// TwinCAT 3 PLC project Main
// ProgramVersion: 3.1.4023.0
// libraries:
//   MotorPositionController, * (Randolf)
//   Tc2_MC2, * (Beckhoff Automation GmbH)
//   Tc2_Standard, * (Beckhoff Automation GmbH)
//   Tc2_System, * (Beckhoff Automation GmbH)
//   Tc3_Module, * (Beckhoff Automation GmbH)
//   VisuDialogs, * (System)
//   VisuSymbols,3.5.10.0,System
// project tree:
//   DUTs/ SensorData.TcDUT
//   / GlobalTextList.TcGTLO, PlcTask.TcTTO (not stored), 视图管理器.TcVMO (not stored)
//   GVLs/ GVL.TcGVL
//   POUs/ MAIN.TcPOU
//   VISUs/ Visualization.TcVIS
// real-time tasks:
//   TASK PlcTask: cycle T#1ms, priority 20, ADS port 350
// motion (NC):
//   TASK NC-Task 1 SAF: cycle T#1ms, priority 4, ADS port 501
//   TASK NC-Task 1 SVB: cycle T#1ms, priority 8, ADS port 511
//   AXIS Axis 1 (id 1)
//     General: UnitName=Degree
//     Dynamic: Acceleration=270, Deceleration=270, Jerk=405
//     Velo: RefSearch=180.759448242188, RefSync=180.759448242188, SlowManual=60, FastManual=120, Fast=18075.9448242188, Maximum=360
//     PositionAreaControl: Enable=false
//     TargetPosControl: Enable=false
//     OtherSettings: AllowMotionCmdToSlave=true
//     encoder EncType=8
//       EncPara: ScaleFactorNumerator=360, ScaleFactorDenominator=1048576, MaxCount=#xffffffff
//     drive DrvType=9
//       DrvPara: MaxCount=#xffffffff, DriveControlDWord=#x00030100
//         Analog: VeloReferenz=360, VeloScale=1.02400649589962, TorqueSetpointScale=10, ScaleFactorActTorque=0.1
//         TimeComp: TaskDelayCycles=1
//     controller CtrType=1
//       CtrPara: PriorControlFactor=1
//         PosDiffControl: Enable=false
//         Observer: BandWidth=20
// I/O:
//   DEVICE Device 3 (EtherCAT), AmsNetId 192.168.137.1.4.1
//     Term 1 (EK1100) [EK1100 EtherCAT Coupler (2A E-Bus)]
//       Term 2 (EL9505) [EL9505 Power supply terminal 5V]
//       Term 3 (EL3356) [EL3356 1Ch. Ana. Input Resistor Bridge Terminal, 16bit, High Precision]
//       Term 5 (EL9011) [EL9011 End Terminal]
//     Drive 4 (AX5106-0000-0203) [AX5106-0000-0203 EtherCAT Drive (SoE, 1 Ch.)]
// variable links:
//   NC-Task 1 SAF/Axes/Axis 1 <-> Device 3 (EtherCAT)/Drive 4 (AX5106-0000-0203)
//     Drive/Inputs/In/nDataIn1 <-> AT/Following distance
//     Drive/Inputs/In/nDcOutputTime <-> InfoData/DcOutputShift
//     Drive/Inputs/In/nState1 <-> AT/Drive status word @bit 8
//     Drive/Inputs/In/nState2 <-> AT/Drive status word
//     Drive/Inputs/In/nState4 @bit 1 <-> WcState/InputToggle
//     Drive/Inputs/In/nState4 <-> WcState/WcState
//     Drive/Outputs/Out/nCtrl1 <-> MDT/Master control word @bit 8
//     Drive/Outputs/Out/nDataOut1 <-> MDT/Position command value
//     Enc/Inputs/In/nDataIn1 <-> AT/Position feedback 1 value
//     Enc/Inputs/In/nDcInputTime <-> InfoData/DcInputShift
//     Enc/Inputs/In/nState4 @bit 1 <-> WcState/InputToggle
//     Enc/Inputs/In/nState4 <-> WcState/WcState
//   Main/Main Instance <-> NC-Task 1 SAF/Axes/Axis 1
//     PlcTask Inputs/GVL.axis1.NcToPlc <-> Outputs/ToPlc
//     PlcTask Outputs/GVL.axis1.PlcToNc <-> Inputs/FromPlc

// ---- DUTs/SensorData.TcDUT
TYPE SensorData :
STRUCT
	force_value_raw AT %I* : REAL;
END_STRUCT
END_TYPE

// ---- GVLs/GVL.TcGVL
{attribute 'qualified_only'}
VAR_GLOBAL
	axis1 : Tc2_MC2.AXIS_REF;
END_VAR

// ---- POUs/MAIN.TcPOU
PROGRAM MAIN
VAR
	motor1 : MotorPositionController;
	motor_param : MotorPositionController.MotorParam;
	motor_data : MotorPositionController.MotorData;
	motor_state : MotorPositionController.MotorState;
	
	sensor_data : SensorData;
END_VAR

motor1(motor_axis:= GVL.axis1, motor_param:= motor_param, motor_data=> motor_data, motor_state=> motor_state);

END_PROGRAM

// ---- GlobalTextList.TcGTLO
TEXTLIST GlobalTextList
  398 = '%5.2f'
  767 = 'Jog反转'
  395 = 'Jog正转'
  15 = 'P2P运动'
  240 = '快速点动'
  151 = '慢速点动'
  924 = '控制操作'
  403 = '期望位置'
  168 = '期望速度'
  199 = '电机Reset'
  433 = '电机位置'
  174 = '电机使能'
  272 = '电机停止'
  942 = '电机故障'
  479 = '电机点动'
  520 = '电机状态'
  743 = '电机运动'
  140 = '电机速度'
  619 = '绝对位置运动'
  522 = '设置零点'
END_TEXTLIST

// ---- VISUs/Visualization.TcVIS
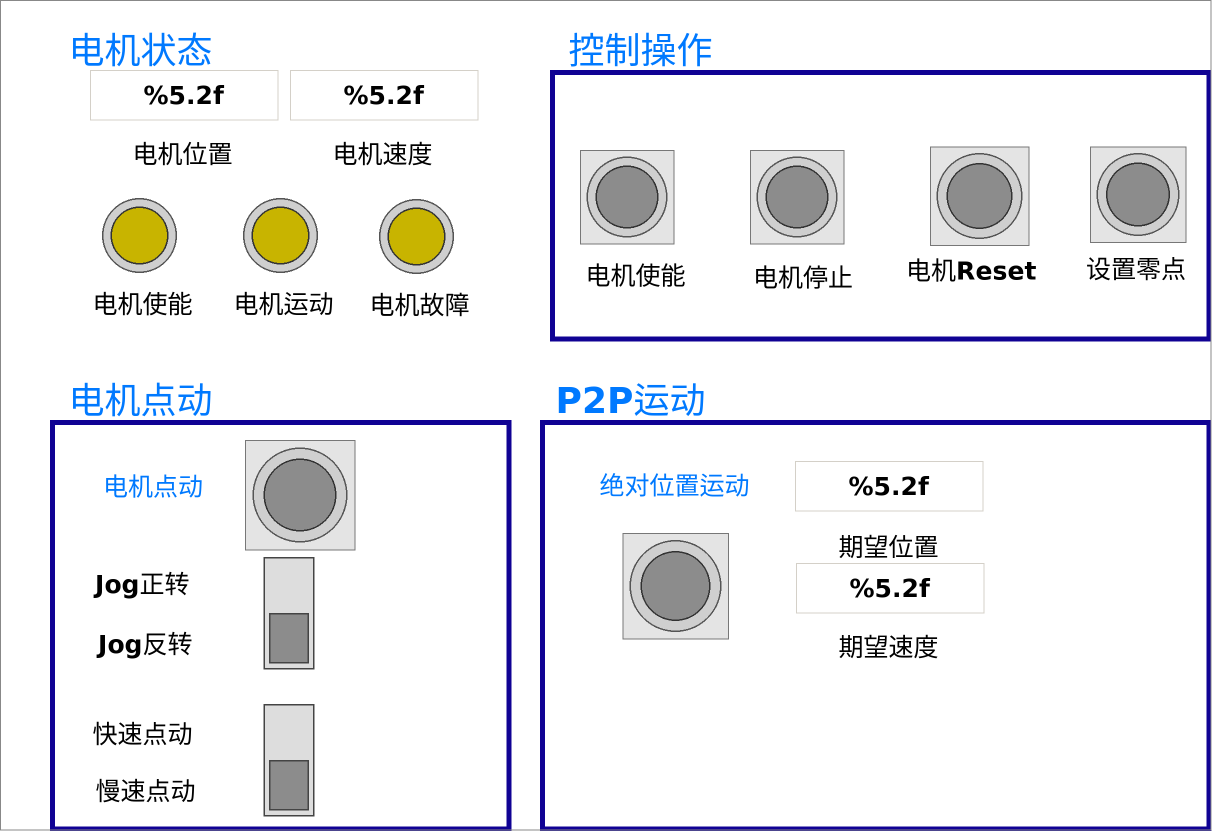
VISUALIZATION Visualization  // 1212x831
    Lamp1 (96,190 87x91), variable: Main.motor_state.is_power_ready, style: Lamp-Lamp1-Yellow
    Label (50,270 185x68), "电机使能"
    Textfield (90,70 188x50), "%5.2f", text variable: Main.motor_data.motor_position
    Label (90,120 185x68), "电机位置"
    Textfield (290,70 188x50), "%5.2f", text variable: Main.motor_data.motor_velocity
    Label (290,120 185x68), "电机速度"
    Lamp1 (237,190 87x91), variable: Main.motor_state.is_motor_moving, style: Lamp-Lamp1-Yellow
    Label (191,270 185x68), "电机运动"
    Label (327,271 185x68), "电机故障"
    Lamp1 (373,191 87x91), variable: Main.motor_state.is_motor_error, style: Lamp-Lamp1-Yellow
    Label (40,20 201x61), "电机状态"
    Rectangle (550,70 661x271)
    Label (560,250 151x51), "电机使能"
    PushSwitchLed (750,140 94x114), variable: Main.motor_param.is_motor_stop, behaviour: TAP, style: Switch-PushSwitchLed-Gray
    Label (730,250 146x55), "电机停止"
    PushSwitchLed (930,140 99x112), variable: Main.motor_param.is_motor_reset, behaviour: TAP, style: Switch-PushSwitchLed-Gray
    Label (890,250 163x41), "电机Reset"
    PushSwitchLed (1090,140 96x109), variable: Main.motor_param.is_set_pos_zero, behaviour: TAP, style: Switch-PushSwitchLed-Gray
    Label (1060,250 152x38), "设置零点"
    PushSwitchLed (580,140 94x114), variable: Main.motor_param.is_motor_power_on, behaviour: TOGGLE, style: Switch-PushSwitchLed-Gray
    Label (540,20 201x61), "控制操作"
    Rectangle (50,420 461x411)
    Label (53,610 185x68), "Jog反转"
    DipSwitch (232,557 114x112), variable: Main.motor_param.jog_direction, behaviour: TOGGLE, style: Switch-DipSwitch-Gray
    Label (50,550 185x68), "Jog正转"
    PushSwitchLed (240,440 120x110), variable: Main.motor_param.is_jog_start, behaviour: TAP, style: Switch-PushSwitchLed-Gray
    Label (90,420 126x133), "电机点动"
    Label (50,700 185x68), "快速点动"
    Label (53,757 185x68), "慢速点动"
    DipSwitch (232,704 114x112), variable: Main.motor_param.jog_mode, behaviour: TOGGLE, style: Switch-DipSwitch-Gray
    Label (40,370 201x61), "电机点动"
    Rectangle (540,420 671x411)
    Textfield (795,461 188x50), "%5.2f", text variable: Main.motor_param.move_abs_target_position
        OnMouseClick: write the text variable via Default
    Label (796,513 185x68), "期望位置"
    Label (796,613 185x68), "期望速度"
    Textfield (796,563 188x50), "%5.2f", text variable: Main.motor_param.move_vel
        OnMouseClick: write the text variable via Default
    PushSwitchLed (616,533 119x106), variable: Main.motor_param.is_motor_moving_abs, behaviour: TAP, style: Switch-PushSwitchLed-Gray
    Label (550,430 249x111), "绝对位置运动"
    Label (530,370 201x61), "P2P运动"
END_VISUALIZATION
